HMI tags "Default tag table"
   "Clock_Byte" : Byte = PLC Clock_Byte AT %MB0, 100 ms
   "HMI_screenNumber" : Int = PLC HMI.screenNumber AT %DB1.DBW0, 100 ms
   "HMI_barcode" : Barcode Screen = PLC HMI.barcode AT %DB1.DBW0, 100 ms
   "HMI_partCall_current{0}" : Table Row = PLC HMI.partCall.current[0], 100 ms
   "HMI_partCall_current{1}" : Table Row = PLC HMI.partCall.current[1], 100 ms
   "HMI_partCall_current{2}" : Table Row = PLC HMI.partCall.current[2], 100 ms
   "HMI_partCall_current{3}" : Table Row = PLC HMI.partCall.current[3], 100 ms
   "HMI_partCall_current{4}" : Table Row = PLC HMI.partCall.current[4], 100 ms
   "HMI_partCall_current{5}" : Table Row = PLC HMI.partCall.current[5], 100 ms
   "HMI_partCall_current{6}" : Table Row = PLC HMI.partCall.current[6], 100 ms
   "HMI_partCall_current{7}" : Table Row = PLC HMI.partCall.current[7], 100 ms
   "HMI_partCall_current{8}" : Table Row = PLC HMI.partCall.current[8], 100 ms
   "HMI_partCall_current{9}" : Table Row = PLC HMI.partCall.current[9], 100 ms
   "HMI_partCall_current{10}" : Table Row = PLC HMI.partCall.current[10], 100 ms
   "HMI_settings_current_stations_selectBtns{0}" : PB Data: Text Label = PLC HMI.settings.current.stations.selectBtns[0], 100 ms
   "HMI_settings_current_stations_selectBtns{1}" : PB Data: Text Label = PLC HMI.settings.current.stations.selectBtns[1], 100 ms
   "HMI_settings_current_stations_selectBtns{2}" : PB Data: Text Label = PLC HMI.settings.current.stations.selectBtns[2], 100 ms
   "HMI_settings_current_stations_selectBtns{3}" : PB Data: Text Label = PLC HMI.settings.current.stations.selectBtns[3], 100 ms
   "HMI_settings_current_stations_selectBtns{4}" : PB Data: Text Label = PLC HMI.settings.current.stations.selectBtns[4], 100 ms
   "HMI_settings_current_stations_selectBtns{5}" : PB Data: Text Label = PLC HMI.settings.current.stations.selectBtns[5], 100 ms
   "HMI_settings_current_stations_selectBtns{6}" : PB Data: Text Label = PLC HMI.settings.current.stations.selectBtns[6], 100 ms
   "HMI_settings_current_stations_selectBtns{7}" : PB Data: Text Label = PLC HMI.settings.current.stations.selectBtns[7], 100 ms
   "HMI_settings_current_stations_selectBtns{8}" : PB Data: Text Label = PLC HMI.settings.current.stations.selectBtns[8], 100 ms
   "HMI_settings_current_stations_selectBtns{9}" : PB Data: Text Label = PLC HMI.settings.current.stations.selectBtns[9], 100 ms
   "HMI_settings_current_stations_selectBtns{10}" : PB Data: Text Label = PLC HMI.settings.current.stations.selectBtns[10], 100 ms
   "HMI_settings_current_stations_selectBtns{11}" : PB Data: Text Label = PLC HMI.settings.current.stations.selectBtns[11], 100 ms
   "HMI_settings_current_kp8_buttons{0}" : PB Data: Text Label = PLC HMI.settings.current.kp8.buttons[0], 100 ms
   "HMI_settings_current_kp8_buttons{7}" : PB Data: Text Label = PLC HMI.settings.current.kp8.buttons[7], 100 ms
   "HMI_settings_current_kp8_buttons{3}" : PB Data: Text Label = PLC HMI.settings.current.kp8.buttons[3], 100 ms
   "HMI_settings_current_kp8_buttons{6}" : PB Data: Text Label = PLC HMI.settings.current.kp8.buttons[6], 100 ms
   "HMI_settings_current_kp8_buttons{2}" : PB Data: Text Label = PLC HMI.settings.current.kp8.buttons[2], 100 ms
   "HMI_settings_current_kp8_buttons{5}" : PB Data: Text Label = PLC HMI.settings.current.kp8.buttons[5], 100 ms
   "HMI_settings_current_kp8_buttons{1}" : PB Data: Text Label = PLC HMI.settings.current.kp8.buttons[1], 100 ms
   "HMI_settings_current_kp8_buttons{4}" : PB Data: Text Label = PLC HMI.settings.current.kp8.buttons[4], 100 ms
   "HMI_settings_current_stations_selCount" : Int = PLC HMI.settings.current.stations.selCount, 100 ms
   "HMI_settings_current_viewingStation_btns{0}" : Station Assignment: Button Details = PLC HMI.settings.current.viewingStation.btns[0], 100 ms
   "HMI_settings_current_viewingStation_btns{1}" : Station Assignment: Button Details = PLC HMI.settings.current.viewingStation.btns[1], 100 ms
   "HMI_settings_current_viewingStation_btns{2}" : Station Assignment: Button Details = PLC HMI.settings.current.viewingStation.btns[2], 100 ms
   "HMI_settings_current_viewingStation_btns{3}" : Station Assignment: Button Details = PLC HMI.settings.current.viewingStation.btns[3], 100 ms
   "HMI_settings_current_viewingStation_btns{4}" : Station Assignment: Button Details = PLC HMI.settings.current.viewingStation.btns[4], 100 ms
   "HMI_settings_current_viewingStation_btns{5}" : Station Assignment: Button Details = PLC HMI.settings.current.viewingStation.btns[5], 100 ms
   "HMI_settings_current_viewingStation_previous" : PB Data: Graphic/Text List = PLC HMI.settings.current.viewingStation.previous, 100 ms
   "HMI_settings_current_viewingStation_next" : PB Data: Graphic/Text List = PLC HMI.settings.current.viewingStation.next, 100 ms
   "HMI_settings_current_stations_selectAll" : PB Data: Text Label = PLC HMI.settings.current.stations.selectAll, 100 ms
   "HMI_settings_current_partNumber_assign" : PB Data: Text Label = PLC HMI.settings.current.partNumber.assign, 100 ms
   "HMI_settings_current_partNumber_ioField" : IO Field Data: Part Number = PLC HMI.settings.current.partNumber.ioField, 100 ms
   "HMI_settings_current_alotted_assign" : PB Data: Text Label = PLC HMI.settings.current.alotted.assign, 100 ms
   "HMI_settings_current_alotted_ioField" : IO Field Data: Timers = PLC HMI.settings.current.alotted.ioField, 100 ms
   "HMI_settings_current_critical_assign" : PB Data: Text Label = PLC HMI.settings.current.critical.assign, 100 ms
   "HMI_settings_current_critical_ioField" : IO Field Data: Timers = PLC HMI.settings.current.critical.ioField, 100 ms
   "HMI_settings_current_kp8_selectButtons" : PB Data: Text Label = PLC HMI.settings.current.kp8.selectButtons, 100 ms
   "HMI_settings_current_viewingStation_dzData" : Drop Zone Data = PLC HMI.settings.current.viewingStation.dzData, 100 ms
   "HMI_settings_current_viewingStation_lineData" : Line Label Data = PLC HMI.settings.current.viewingStation.lineData, 100 ms
   "HMI_settings_current_stations_prevGroup" : PB Data: Graphic/Text List = PLC HMI.settings.current.stations.prevGroup, 100 ms
   "HMI_settings_current_stations_nextGroup" : PB Data: Graphic/Text List = PLC HMI.settings.current.stations.nextGroup, 100 ms
   "HMI_settings_current_viewingStation_name" : WString[20] = PLC HMI.settings.current.viewingStation.name, 100 ms

text list "Station Selection Single": 0 'Select a Station to View'; 1 'Assignments'

screen "1 PART CALL" 1366x768
   on GenerateScreen: SetTag("HMI_screenNumber", 1)
   Rectangle "Nav Panel 02" at 682,700 size 684x68
      Appearance <- "HMI_screenNumber"
   Rectangle "Nav Panel 01" at 0,700 size 685x68
      Appearance <- "HMI_screenNumber"
   Rectangle "Nav Panel 03 Top Border Hide" at 685,700 size 678x3
      Visibility <- "HMI_screenNumber"
   Rectangle "Nav Panel 01 Top Border Hide" at 3,700 size 679x3
      Visibility <- "HMI_screenNumber"
   Button "Settings Screen" at 683,700 size 683x68; TextOff 'SETTINGS'; Authorization "User administration"
      on Release: ActivateScreen("2 SETTINGS", 0)
   Button "Part Call Screen" at 0,700 size 683x68; TextOff 'PART CALL'
      on Release: ActivateScreen("1 PART CALL", 0)
   TextField "Header Line" at 32,32 size 216x53; Text 'LINE'
   TextField "Header Drop Zone" at 238,32 size 236x53; Text 'DROP ZONE'
   TextField "Header Part Number" at 474,32 size 648x53; Text 'PART NUMBER'
   TextField "Header Time" at 1112,32 size 222x53; Text 'TIME'
   ScreenModuleView "TableRow00" at 27,90 size 1312x52; ScreenModuleType ""
      Guid_{11997190-27688} <- "HMI_partCall_current{0}"
   ScreenModuleView "TableRow01" at 27,142 size 1312x52; ScreenModuleType ""
      Guid_{11997190-27688} <- "HMI_partCall_current{1}"
   ScreenModuleView "TableRow02" at 27,194 size 1312x52; ScreenModuleType ""
      Guid_{11997190-27688} <- "HMI_partCall_current{2}"
   ScreenModuleView "TableRow03" at 27,246 size 1312x52; ScreenModuleType ""
      Guid_{11997190-27688} <- "HMI_partCall_current{3}"
   ScreenModuleView "TableRow04" at 27,298 size 1312x52; ScreenModuleType ""
      Guid_{11997190-27688} <- "HMI_partCall_current{4}"
   ScreenModuleView "TableRow05" at 27,350 size 1312x52; ScreenModuleType ""
      Guid_{11997190-27688} <- "HMI_partCall_current{5}"
   ScreenModuleView "TableRow06" at 27,402 size 1312x52; ScreenModuleType ""
      Guid_{11997190-27688} <- "HMI_partCall_current{6}"
   ScreenModuleView "TableRow07" at 27,454 size 1312x52; ScreenModuleType ""
      Guid_{11997190-27688} <- "HMI_partCall_current{7}"
   ScreenModuleView "TableRow08" at 27,506 size 1312x52; ScreenModuleType ""
      Guid_{11997190-27688} <- "HMI_partCall_current{8}"
   ScreenModuleView "TableRow09" at 27,558 size 1312x52; ScreenModuleType ""
      Guid_{11997190-27688} <- "HMI_partCall_current{9}"
   ScreenModuleView "TableRow10" at 27,610 size 1312x52; ScreenModuleType ""
      Guid_{11997190-27688} <- "HMI_partCall_current{10}"

screen "2 SETTINGS" 1366x768
   on GenerateScreen: SetTag("HMI_screenNumber", 2)
   Rectangle "Part Call Nave Panel" at 0,700 size 685x68
      Appearance <- "HMI_screenNumber"
   Rectangle "Settings Nav Panel" at 682,700 size 684x68
      Appearance <- "HMI_screenNumber"
   Rectangle "Part Call Top Border Hide" at 3,700 size 679x3
      Visibility <- "HMI_screenNumber"
   Rectangle "Settings Top Border Hide" at 685,700 size 678x3
      Visibility <- "HMI_screenNumber"
   Button "Part Call Screen" at 0,700 size 683x68; TextOff 'PART CALL'
      on Release: ActivateScreen("1 PART CALL", 0)
   Button "Settings Screen" at 683,700 size 683x68; TextOff 'SETTINGS'
      on Release: ActivateScreen("2 SETTINGS", 0)
   Rectangle "Station Assignment Table BG Full" at 793,40 size 533x630
      Visibility <- "HMI_settings_current_stations_selCount"
   TextField "Current Station Single" at 803,50 size 513x45; Text 'Text'
      Visibility <- "HMI_settings_current_stations_selCount"
   TextField "Hide Line and Drop Zone Multi" at 803,101 size 513x40; Text 'select single station for Line and Drop Zone'
      Visibility <- "HMI_settings_current_stations_selCount"
   GraphicView "KP8 Image" at 496,247 size 275x412; Picture "kp8 image"
   Rectangle "Station Assignment Table BG Mini" at 793,40 size 533x65
      Visibility <- "HMI_settings_current_stations_selCount"
   ScreenModuleView "PB: Set PN" at 50,50 size 414x45; Guid_{11997190-63616} 'Assign Part Number'; ScreenModuleType ""
      Guid_{11997190-63605} <- "HMI_settings_current_partNumber_assign"
   ScreenModuleView "PN IO Field" at 50,100 size 414x50; ScreenModuleType ""
      Guid_{11997190-63113} <- "HMI_settings_current_partNumber_ioField"
   ScreenModuleView "PB: Set Allotted" at 494,50 size 137x45; Guid_{11997190-63616} 'Allotted'; ScreenModuleType ""
      Guid_{11997190-63605} <- "HMI_settings_current_alotted_assign"
   ScreenModuleView "PB: Set Critical" at 636,50 size 137x45; Guid_{11997190-63616} 'Crititcal'; ScreenModuleType ""
      Guid_{11997190-63605} <- "HMI_settings_current_critical_assign"
   ScreenModuleView "Alotted Time IO Field" at 494,100 size 137x50; ScreenModuleType ""
      Guid_{11997190-63269} <- "HMI_settings_current_alotted_ioField"
   ScreenModuleView "Critical Time IO Field" at 636,100 size 137x50; ScreenModuleType ""
      Guid_{11997190-63269} <- "HMI_settings_current_critical_ioField"
   ScreenModuleView "PB: Select KP8 Buttons" at 493,190 size 284x45; Guid_{11997190-63616} 'Select Buttons'; ScreenModuleType ""
      Guid_{11997190-63605} <- "HMI_settings_current_kp8_selectButtons"
   ScreenModuleView "KP8 00: RESET" at 641,534 size 68x66; ScreenModuleType ""
      Guid_{11997190-57808} <- "HMI_settings_current_kp8_buttons{0}"
   ScreenModuleView "KP8 01" at 641,455 size 68x66; ScreenModuleType ""
      Guid_{11997190-57808} <- "HMI_settings_current_kp8_buttons{1}"
   ScreenModuleView "KP8 02" at 641,379 size 68x66; ScreenModuleType ""
      Guid_{11997190-57808} <- "HMI_settings_current_kp8_buttons{2}"
   ScreenModuleView "KP8 03" at 641,303 size 68x66; ScreenModuleType ""
      Guid_{11997190-57808} <- "HMI_settings_current_kp8_buttons{3}"
   ScreenModuleView "KP8 04: STOP RUNTIME" at 557,534 size 68x66; ScreenModuleType ""
      on Guid_{11997190-59171}: StopRuntime(0)
      Guid_{11997190-57808} <- "HMI_settings_current_kp8_buttons{4}"
   ScreenModuleView "KP8 05" at 557,455 size 68x66; ScreenModuleType ""
      Guid_{11997190-57808} <- "HMI_settings_current_kp8_buttons{5}"
   ScreenModuleView "KP8 06" at 557,379 size 68x66; ScreenModuleType ""
      Guid_{11997190-57808} <- "HMI_settings_current_kp8_buttons{6}"
   ScreenModuleView "KP8 07" at 557,303 size 68x66; ScreenModuleType ""
      Guid_{11997190-57808} <- "HMI_settings_current_kp8_buttons{7}"
   ScreenModuleView "PB: Previous Group" at 50,190 size 65x45; Guid_{11997190-63799} "Graphic_4"; ScreenModuleType ""
      Guid_{11997190-63779} <- "HMI_settings_current_stations_prevGroup"
   ScreenModuleView "PB: Select All Stations" at 120,190 size 274x45; Guid_{11997190-63616} 'Select Stations'; ScreenModuleType ""
      Guid_{11997190-63605} <- "HMI_settings_current_stations_selectAll"
   ScreenModuleView "PB: Next Group" at 399,190 size 65x45; Guid_{11997190-63799} "Graphic_3"; ScreenModuleType ""
      Guid_{11997190-63779} <- "HMI_settings_current_stations_nextGroup"
   ScreenModuleView "Station 00 Select" at 50,240 size 205x65; ScreenModuleType ""
      Guid_{11997190-57808} <- "HMI_settings_current_stations_selectBtns{0}"
   ScreenModuleView "Station 01 Select" at 260,240 size 205x65; ScreenModuleType ""
      Guid_{11997190-57808} <- "HMI_settings_current_stations_selectBtns{1}"
   ScreenModuleView "Station 02 Select" at 50,311 size 205x65; ScreenModuleType ""
      Guid_{11997190-57808} <- "HMI_settings_current_stations_selectBtns{2}"
   ScreenModuleView "Station 03 Select" at 260,311 size 205x65; ScreenModuleType ""
      Guid_{11997190-57808} <- "HMI_settings_current_stations_selectBtns{3}"
   ScreenModuleView "Station 04 Select" at 50,382 size 205x65; ScreenModuleType ""
      Guid_{11997190-57808} <- "HMI_settings_current_stations_selectBtns{4}"
   ScreenModuleView "Station 05 Select" at 260,382 size 205x65; ScreenModuleType ""
      Guid_{11997190-57808} <- "HMI_settings_current_stations_selectBtns{5}"
   ScreenModuleView "Station 06 Select" at 50,453 size 205x65; ScreenModuleType ""
      Guid_{11997190-57808} <- "HMI_settings_current_stations_selectBtns{6}"
   ScreenModuleView "Station 07 Select" at 260,453 size 205x65; ScreenModuleType ""
      Guid_{11997190-57808} <- "HMI_settings_current_stations_selectBtns{7}"
   ScreenModuleView "Station 08 Select" at 50,524 size 205x65; ScreenModuleType ""
      Guid_{11997190-57808} <- "HMI_settings_current_stations_selectBtns{8}"
   ScreenModuleView "Station 09 Select" at 260,524 size 205x65; ScreenModuleType ""
      Guid_{11997190-57808} <- "HMI_settings_current_stations_selectBtns{9}"
   ScreenModuleView "Station 10 Select" at 50,595 size 205x65; ScreenModuleType ""
      Guid_{11997190-57808} <- "HMI_settings_current_stations_selectBtns{10}"
   ScreenModuleView "Station 11 Select" at 260,595 size 205x65; ScreenModuleType ""
      Guid_{11997190-57808} <- "HMI_settings_current_stations_selectBtns{11}"
   ScreenModuleView "Line Label" at 803,101 size 267x40; ScreenModuleType ""
      Guid_{11997190-64598} <- "HMI_settings_current_viewingStation_lineData"
   ScreenModuleView "Drop Zone Label" at 1076,101 size 240x40; ScreenModuleType ""
      Guid_{11997190-64802} <- "HMI_settings_current_viewingStation_dzData"
   ScreenModuleView "PB: Previous Station" at 803,50 size 65x45; Guid_{11997190-63799} "Graphic_1"; ScreenModuleType ""
      Guid_{11997190-63779} <- "HMI_settings_current_viewingStation_previous"
   TextField "Current Station Multi" at 873,50 size 373x45; Text 'Assignments'
      Visibility <- "HMI_settings_current_stations_selCount"
   ScreenModuleView "PB: Next Station" at 1251,50 size 65x45; Guid_{11997190-63799} "Graphic_2"; ScreenModuleType ""
      Guid_{11997190-63779} <- "HMI_settings_current_viewingStation_previous"
   TextField "Button Column Header" at 803,146 size 75x40; Text 'Btn'
      Visibility <- "HMI_settings_current_stations_selCount"
   TextField "Timer Column Header" at 872,146 size 128x40; Text 'Times'
      Visibility <- "HMI_settings_current_stations_selCount"
   TextField "Part Number Column Header" at 993,146 size 323x40; Text 'Part Number'
      Visibility <- "HMI_settings_current_stations_selCount"
   ScreenModuleView "Button 00 Details" at 803,191 size 513x74; ScreenModuleType ""
      Guid_{11997190-60358} <- "HMI_settings_current_viewingStation_btns{0}"
   ScreenModuleView "Button 01 Details" at 803,270 size 513x74; ScreenModuleType ""
      Guid_{11997190-60358} <- "HMI_settings_current_viewingStation_btns{1}"
   ScreenModuleView "Button 02 Details" at 803,349 size 513x74; ScreenModuleType ""
      Guid_{11997190-60358} <- "HMI_settings_current_viewingStation_btns{2}"
   ScreenModuleView "Button 03 Details" at 803,428 size 513x74; ScreenModuleType ""
      Guid_{11997190-60358} <- "HMI_settings_current_viewingStation_btns{3}"
   ScreenModuleView "Button 04 Details" at 803,507 size 513x74; ScreenModuleType ""
      Guid_{11997190-60358} <- "HMI_settings_current_viewingStation_btns{4}"
   ScreenModuleView "Button 05 Details" at 803,586 size 513x74; ScreenModuleType ""
      Guid_{11997190-60358} <- "HMI_settings_current_viewingStation_btns{5}"

screen "3 BARCODE" 1366x768
   on GenerateScreen: SetTag("HMI_screenNumber", 3)
   Rectangle "Nav Panel 02" at 682,700 size 684x68
      Appearance <- "HMI_screenNumber"
   Rectangle "Nav Panel 01" at 0,700 size 685x68
      Appearance <- "HMI_screenNumber"
   Rectangle "Nav Panel 03 Top Border Hide" at 685,700 size 678x3
      Visibility <- "HMI_screenNumber"
   Rectangle "Nav Panel 01 Top Border Hide" at 3,700 size 679x3
      Visibility <- "HMI_screenNumber"
   Button "Settings Screen" at 683,700 size 683x68; TextOff 'SETTINGS'; Authorization "User administration"
      on Release: ActivateScreen("2 SETTINGS", 0)
   Button "Part Call Screen" at 0,700 size 683x68; TextOff 'PART CALL'
      on Release: ActivateScreen("1 PART CALL", 0)
   Button "btCancel" at 685,431 size 649x68; TextOff 'CANCEL'
      on Release: ActivateScreen("1 PART CALL", 0)
   Button "btPartOrdered" at 32,431 size 648x68; TextOff 'ORDERED'
      on Release: SetBit("ordered"); ActivateScreen("1 PART CALL", 0)
   TextField "tfBarcodeDisplay" at 32,220 size 1302x206; Text 'Text'
   TextField "tfPartNumberDisplay" at 32,160 size 1302x53; Text 'BARCODE FOR PART NUMBER'
*)

(* ===== HMI "HMI_RT_2" =====
connection "HMI_Connection_3": ETHERNET, S7_1500_OMS

HMI tags "Default tag table"
   "Clock_0.5Hz" : Bool = PLC "Clock_0.5Hz" AT %M0.7, 100 ms
   "LED Sign_request_row{0}" : Table Row = PLC "LED Sign".request.row[0], 1 s
   "LED Sign_request_row{1}" : Table Row = PLC "LED Sign".request.row[1], 1 s
   "LED Sign_request_row{2}" : Table Row = PLC "LED Sign".request.row[2], 1 s
   "LED Sign_request_row{3}" : Table Row = PLC "LED Sign".request.row[3], 1 s
   "LED Sign_request_row{4}" : Table Row = PLC "LED Sign".request.row[4], 1 s
   "LED Sign_request_row{5}" : Table Row = PLC "LED Sign".request.row[5], 1 s
   "LED Sign_request_row{6}" : Table Row = PLC "LED Sign".request.row[6], 1 s
   "LED Sign_request_row{7}" : Table Row = PLC "LED Sign".request.row[7], 1 s
   "LED Sign_request_row{8}" : Table Row = PLC "LED Sign".request.row[8], 1 s
   "LED Sign_request_row{9}" : Table Row = PLC "LED Sign".request.row[9], 1 s
   "LED Sign_request_row{10}" : Table Row = PLC "LED Sign".request.row[10], 1 s
   "LED Sign_request_row{11}" : Table Row = PLC "LED Sign".request.row[11], 1 s

screen "1 PART CALL" 1024x768
   Rectangle "Connection Status" at 1,196 size 894x1
      Appearance <- "Clock_0.5Hz"
   ScreenModuleView "R0C0" at 6,9 size 440x28; ScreenModuleType ""
      Guid_{11997190-27688} <- "LED Sign_request_row{0}"
   ScreenModuleView "R1C0" at 6,39 size 440x28; ScreenModuleType ""
      Guid_{11997190-27688} <- "LED Sign_request_row{1}"
   ScreenModuleView "R2C0" at 6,69 size 440x28; ScreenModuleType ""
      Guid_{11997190-27688} <- "LED Sign_request_row{2}"
   ScreenModuleView "R3C0" at 6,99 size 440x28; ScreenModuleType ""
      Guid_{11997190-27688} <- "LED Sign_request_row{3}"
   ScreenModuleView "R4C0" at 6,128 size 440x28; ScreenModuleType ""
      Guid_{11997190-27688} <- "LED Sign_request_row{4}"
   ScreenModuleView "R5C0" at 6,158 size 440x28; ScreenModuleType ""
      Guid_{11997190-27688} <- "LED Sign_request_row{5}"
   ScreenModuleView "R0C1" at 455,9 size 438x28; ScreenModuleType ""
      Guid_{11997190-27688} <- "LED Sign_request_row{6}"
   ScreenModuleView "R1C1" at 455,39 size 438x28; ScreenModuleType ""
      Guid_{11997190-27688} <- "LED Sign_request_row{7}"
   ScreenModuleView "R2C1" at 454,69 size 440x28; ScreenModuleType ""
      Guid_{11997190-27688} <- "LED Sign_request_row{8}"
   ScreenModuleView "R3C1" at 454,99 size 440x28; ScreenModuleType ""
      Guid_{11997190-27688} <- "LED Sign_request_row{9}"
   ScreenModuleView "R4C1" at 454,128 size 440x28; ScreenModuleType ""
      Guid_{11997190-27688} <- "LED Sign_request_row{10}"
   ScreenModuleView "R5C1" at 454,158 size 440x28; ScreenModuleType ""
      Guid_{11997190-27688} <- "LED Sign_request_row{11}"
*)

(* ===== HMI "HMI_RT_1" =====
system functions are stored by id; their names below are inferred from use

ScreenModuleEditorView "Table Row" 1312x52
   TextField "tfLine" at 5,1 size 216x48; Text 'Text'
      Visibility <- "interface.tfLine.visibility"
      Appearance <- "interface.tfLine.animator"
   TextField "tfTime" at 1085,1 size 222x48; Text 'Text'
      Appearance <- "interface.tfTime.animator"
      Visibility <- "interface.tfTime.visibility"
   TextField "tfDropZone" at 211,1 size 236x48; Text 'Text'
      Appearance <- "interface.tfDropZone.animator"
      Visibility <- "interface.tfDropZone.visibility"
   TextField "tfPartNumber" at 445,1 size 650x48; Text 'Text'
      Appearance <- "interface.tfPartNumber.animator"
      Visibility <- "interface.tfPartNumber.visibility"
   Button "pbSelect" at 0,0 size 1312x52; TextOff 'Text'
      Visibility <- "interface.pbSelection.visibility"
      on Press: SetBit("interface.pbSelection.request")
      on Release: ResetBit("interface.pbSelection.request")
   Rectangle "rtBackground" at 0,0 size 1312x52
      Visibility <- "interface.rtBackground.visibility"
*)

(* ===== HMI "HMI_RT_1" =====
system functions are stored by id; their names below are inferred from use

ScreenModuleEditorView "Table Row" 1312x52
   TextField "tfLine" at 5,1 size 216x48; Text 'Text'
      Visibility <- "interface.tfLine.visibility"
      Appearance <- "interface.tfLine.animator"
   TextField "tfTime" at 1085,1 size 222x48; Text 'Text'
      Visibility <- "interface.tfTime.visibility"
      Appearance <- "interface.tfTime.animator"
   TextField "tfDropZone" at 211,1 size 236x48; Text 'Text'
      Visibility <- "interface.tfDropZone.visibility"
      Appearance <- "interface.tfDropZone.animator"
   TextField "tfPartNumber" at 445,1 size 650x48; Text 'Text'
      Visibility <- "interface.tfPartNumber.visibility"
      Appearance <- "interface.tfPartNumber.animator"
   Button "pbSelect" at 0,0 size 1312x52; TextOff 'Text'
      on Release: ResetBit("interface.pbSelection.request")
      on Press: SetBit("interface.pbSelection.request")
      Visibility <- "interface.pbSelection.visibility"
   Rectangle "rtBackground" at 0,0 size 1312x52
      Visibility <- "interface.rtBackground.visibility"
*)

(* ===== HMI "HMI_RT_1" =====
system functions are stored by id; their names below are inferred from use

ScreenModuleEditorView "Table Row" 1312x52
   TextField "tfLine" at 5,1 size 216x48; Text 'Text'
      Visibility <- "interface.tfLine.visibility"
      Appearance <- "interface.tfLine.animator"
   TextField "tfTime" at 1085,1 size 222x48; Text 'Text'
      Visibility <- "interface.tfTime.visibility"
      Appearance <- "interface.tfTime.animator"
   TextField "tfDropZone" at 211,1 size 236x48; Text 'Text'
      Visibility <- "interface.tfDropZone.visibility"
      Appearance <- "interface.tfDropZone.animator"
   TextField "tfPartNumber" at 445,1 size 650x48; Text 'Text'
      Visibility <- "interface.tfPartNumber.visibility"
      Appearance <- "interface.tfPartNumber.animator"
   Button "pbSelect" at 0,0 size 1312x52; TextOff 'Text'
      on Release: ResetBit("interface.pbSelection.request")
      on Press: SetBit("interface.pbSelection.request")
      Visibility <- "interface.pbSelection.visibility"
   Rectangle "rtBackground" at 0,0 size 1312x52
      Visibility <- "interface.rtBackground.visibility"
*)

(* ===== HMI "HMI_RT_1" =====
system functions are stored by id; their names below are inferred from use

ScreenModuleEditorView "Table Row" 1312x52
   TextField "tfLine" at 5,1 size 216x48; Text 'Text'
      Visibility <- "interface.tfLine.visibility"
      Appearance <- "interface.tfLine.animator"
   TextField "tfTime" at 1085,1 size 222x48; Text 'Text'
      Visibility <- "interface.tfTime.visibility"
      Appearance <- "interface.tfTime.animator"
   TextField "tfDropZone" at 211,1 size 236x48; Text 'Text'
      Visibility <- "interface.tfDropZone.visibility"
      Appearance <- "interface.tfDropZone.animator"
   TextField "tfPartNumber" at 445,1 size 650x48; Text 'Text'
      Visibility <- "interface.tfPartNumber.visibility"
      Appearance <- "interface.tfPartNumber.animator"
   Button "pbSelect" at 0,0 size 1312x52; TextOff 'Text'
      on Release: ResetBit("interface.pbSelection.request")
      on Press: SetBit("interface.pbSelection.request")
      Visibility <- "interface.pbSelection.visibility"
   Rectangle "rtBackground" at 0,0 size 1312x52
      Visibility <- "interface.rtBackground.visibility"
*)

(* ===== HMI "HMI_RT_1" =====
system functions are stored by id; their names below are inferred from use

ScreenModuleEditorView "Table Row" 1312x52
   TextField "tfLine" at 5,1 size 216x48; Text 'Text'
      Visibility <- "interface.tfLine.visibility"
      Appearance <- "interface.tfLine.animator"
   TextField "tfTime" at 1085,1 size 222x48; Text 'Text'
      Visibility <- "interface.tfTime.visibility"
      Appearance <- "interface.tfTime.animator"
   TextField "tfDropZone" at 211,1 size 236x48; Text 'Text'
      Visibility <- "interface.tfDropZone.visibility"
      Appearance <- "interface.tfDropZone.animator"
   TextField "tfPartNumber" at 445,1 size 650x48; Text 'Text'
      Visibility <- "interface.tfPartNumber.visibility"
      Appearance <- "interface.tfPartNumber.animator"
   Button "pbSelect" at 0,0 size 1312x52; TextOff 'Text'
      on Release: ResetBit("interface.pbSelection.request")
      on Press: SetBit("interface.pbSelection.request")
      Visibility <- "interface.pbSelection.visibility"
   Rectangle "rtBackground" at 0,0 size 1312x52
      Visibility <- "interface.rtBackground.visibility"
*)

(* ===== HMI "HMI_RT_1" =====
system functions are stored by id; their names below are inferred from use

ScreenModuleEditorView "LED Row" 1312x52
   TextField "tfLine" at 5,1 size 216x48; Text 'Text'
      Visibility <- "interface.tfLine.visibility"
      Appearance <- "interface.tfLine.animator"
   TextField "tfTime" at 1085,1 size 222x48; Text 'Text'
      Visibility <- "interface.tfTime.visibility"
      Appearance <- "interface.tfTime.animator"
   TextField "tfDropZone" at 211,1 size 236x48; Text 'Text'
      Visibility <- "interface.tfDropZone.visibility"
      Appearance <- "interface.tfDropZone.animator"
   TextField "tfPartNumber" at 445,1 size 650x48; Text 'Text'
      Visibility <- "interface.tfPartNumber.visibility"
      Appearance <- "interface.tfPartNumber.animator"
   Button "pbSelect" at 0,0 size 1312x52; TextOff 'Text'
      on Release: ResetBit("interface.pbSelection.request")
      on Press: SetBit("interface.pbSelection.request")
      Visibility <- "interface.pbSelection.visibility"
   Rectangle "rtBackground" at 0,0 size 1312x52
      Visibility <- "interface.rtBackground.visibility"
*)

(* ===== HMI "HMI_RT_1" =====
system functions are stored by id; their names below are inferred from use

ScreenModuleEditorView "LED Row" 440x28
   TextField "tfLine" at 0,0 size 110x28; Text 'Text'
      Visibility <- "interface.tfLine.visibility"
      Appearance <- "interface.tfLine.animator"
   TextField "tfTime" at 349,0 size 91x28; Text 'Text'
      Visibility <- "interface.tfTime.visibility"
      Appearance <- "interface.tfTime.animator"
   TextField "tfDropZone" at 105,0 size 42x28; Text 'Text'
      Visibility <- "interface.tfDropZone.visibility"
      Appearance <- "interface.tfDropZone.animator"
   TextField "tfDLPartNumber" at 146,0 size 209x28; Text 'Text'
      Appearance <- "interface.tfPartNumber.animator"
      Visibility <- "interface.tfPartNumber.count"
   Button "pbSelect" at 0,0 size 440x28; TextOff 'Text'
      on Release: ResetBit("interface.pbSelection.request")
      on Press: SetBit("interface.pbSelection.request")
      Visibility <- "interface.pbSelection.visibility"
   Rectangle "rtBackground" at 0,0 size 440x28
      Visibility <- "interface.rtBackground.visibility"
   TextField "tfSLPartNumber" at 146,0 size 209x28; Text 'Text'
      Appearance <- "interface.tfPartNumber.animator"
      Visibility <- "interface.tfPartNumber.count"
*)

(* ===== HMI "HMI_RT_1" =====
system functions are stored by id; their names below are inferred from use

ScreenModuleEditorView "Table Row" 1312x52
   TextField "tfLine" at 5,1 size 216x48; Text 'Text'
      Visibility <- "interface.tfLine.visibility"
      Appearance <- "interface.tfLine.animator"
   TextField "tfTime" at 1085,1 size 222x48; Text 'Text'
      Visibility <- "interface.tfTime.visibility"
      Appearance <- "interface.tfTime.animator"
   TextField "tfDropZone" at 211,1 size 236x48; Text 'Text'
      Visibility <- "interface.tfDropZone.visibility"
      Appearance <- "interface.tfDropZone.animator"
   TextField "tfSLPartNumber" at 445,1 size 650x48; Text 'Text'
      Appearance <- "interface.tfPartNumber.animator"
      Visibility <- "interface.tfPartNumber.count"
   Button "pbSelect" at 0,0 size 1312x52; TextOff 'Text'
      on Release: ResetBit("interface.pbSelection.request")
      on Press: SetBit("interface.pbSelection.request")
      Visibility <- "interface.pbSelection.visibility"
   Rectangle "rtBackground" at 0,0 size 1312x52
      Visibility <- "interface.rtBackground.visibility"
   TextField "tfDLPartNumber" at 445,1 size 650x48; Text 'Text'
      Appearance <- "interface.tfPartNumber.animator"
      Visibility <- "interface.tfPartNumber.count"
*)

(* ===== HMI "HMI_RT_1" =====

ScreenModuleEditorView "LED Row" 440x28
   TextField "tfLine" at 0,0 size 110x28; Text 'Text'
      Visibility <- "interface.tfLine.visibility"
      Appearance <- "interface.tfLine.animator"
   TextField "tfTime" at 349,0 size 91x28; Text 'Text'
      Visibility <- "interface.tfTime.visibility"
      Appearance <- "interface.tfTime.animator"
   TextField "tfDropZone" at 105,0 size 42x28; Text 'Text'
      Visibility <- "interface.tfDropZone.visibility"
      Appearance <- "interface.tfDropZone.animator"
   TextField "tfSLPartNumber" at 146,0 size 209x28; Text 'Text'
      Visibility <- "interface.tfPartNumber.count"
      Appearance <- "interface.tfPartNumber.animator"
   TextField "tfDLPartNumber" at 146,0 size 209x28; Text 'Text'
      Visibility <- "interface.tfPartNumber.count"
      Appearance <- "interface.tfPartNumber.animator"
*)

(* ===== HMI "HMI_RT_1" =====
system functions are stored by id; their names below are inferred from use

ScreenModuleEditorView "Table Row" 1312x52
   TextField "tfLine" at 5,1 size 216x48; Text 'Text'
      Visibility <- "interface.tfLine.visibility"
      Appearance <- "interface.tfLine.animator"
   TextField "tfTime" at 1085,1 size 222x48; Text 'Text'
      Visibility <- "interface.tfTime.visibility"
      Appearance <- "interface.tfTime.animator"
   TextField "tfDropZone" at 211,1 size 236x48; Text 'Text'
      Visibility <- "interface.tfDropZone.visibility"
      Appearance <- "interface.tfDropZone.animator"
   TextField "tfSLPartNumber" at 445,1 size 650x48; Text 'Text'
      Visibility <- "interface.tfPartNumber.count"
      Appearance <- "interface.tfPartNumber.animator"
   Button "pbSelect" at 0,0 size 1312x52; TextOff 'Text'
      on Release: ResetBit("interface.pbSelection.request")
      on Press: SetBit("interface.pbSelection.request")
      Visibility <- "interface.pbSelection.visibility"
   Rectangle "rtBackground" at 0,0 size 1312x52
      Visibility <- "interface.rtBackground.visibility"
   TextField "tfDLPartNumber" at 445,1 size 650x48; Text 'Text'
      Visibility <- "interface.tfPartNumber.count"
      Appearance <- "interface.tfPartNumber.animator"
*)

(* ===== HMI "HMI_RT_1" =====
system functions are stored by id; their names below are inferred from use

ScreenModuleEditorView "PB: Station Select (Text Label)" 205x65
   Button "Station Select" at 0,0 size 205x65; TextOff 'Text'
      on Press: function_b14e0dd5("Interface.actuate", 0)
      Appearance <- "Interface.animate"
*)

(* ===== HMI "HMI_RT_1" =====
system functions are stored by id; their names below are inferred from use

ScreenModuleEditorView "PB: KP8 Button Select (Text Label)" 205x65
   Button "Station Select" at 0,0 size 205x65; TextOff 'Text'
      on Press: function_b14e0dd5("Interface.actuate", 0)
      Appearance <- "Interface.animate"
*)

(* ===== HMI "HMI_RT_1" =====
system functions are stored by id; their names below are inferred from use

ScreenModuleEditorView "PB: KP8 Button Select (Text Label)" 68x66
   Button "Station Select" at 0,0 size 68x66; TextOff 'Text'
      on Press: function_b14e0dd5("Interface.actuate", 0)
      Appearance <- "Interface.animate"
*)

(* ===== HMI "HMI_RT_1" =====
system functions are stored by id; their names below are inferred from use

ScreenModuleEditorView "PB: KP8 Stop Runtime (Text Label)" 68x66
   Button "Station Select" at 0,0 size 68x66; TextOff 'Text'
      on Press: function_b14e0dd5("Interface.actuate", 0)
      Appearance <- "Interface.animate"
*)

(* ===== HMI "HMI_RT_1" =====

ScreenModuleEditorView "PB: KP8 Stop Runtime (Text Label)" 68x66
   Button "Station Select" at 0,0 size 68x66; TextOff 'NOT USED'
      Appearance <- "Interface.animate"
*)

(* ===== HMI "HMI_RT_1" =====

ScreenModuleEditorView "PB: KP8 Stop Runtime (Text Label)" 68x66
   Button "Station Select" at 0,0 size 68x66; TextOff 'NOT USED'
      Appearance <- "Interface.animate"
*)

(* ===== HMI "HMI_RT_1" =====
system functions are stored by id; their names below are inferred from use

ScreenModuleEditorView "Station Assignment: Button Details" 513x74
   TextField "Button Label" at 0,0 size 75x74; Text 'Text'
      Appearance <- "Interface.label.animate"
      Visibility <- "Interface.label.animate"
   TextField "Critical Time" at 70,37 size 122x37; Text 'Text'
      Appearance <- "Interface.critical.animate"
      Visibility <- "Interface.critical.animate"
   TextField "Alloted Time" at 70,0 size 122x38; Text 'Text'
      Appearance <- "Interface.alloted.animate"
      Visibility <- "Interface.alloted.animate"
   TextField "Part Number" at 185,0 size 328x74; Text 'Text'
      Appearance <- "Interface.partNumber.animate"
      Visibility <- "Interface.partNumber.animate"
   Button "Select PB" at 0,0 size 513x74; TextOff 'Text'
      on Press: function_b14e0dd5("Interface.select.actuate", 0)
      Visibility <- "Interface.select.animate"
      ObjectEnable <- "Interface.select.animate"
*)

(* ===== HMI "HMI_RT_1" =====
system functions are stored by id; their names below are inferred from use

ScreenModuleEditorView "IO Field: Part Number" 414x50
   IOField "PN Entry Field" at 0,0 size 414x50; FormatPattern ????????????????????????????????????????
      on OnFinishInput: SetBit("Interface.inputFinished")
      ObjectEnable <- "Interface.animate"
      Appearance <- "Interface.animate"
      ProcessValue <- "Interface.value"
*)

(* ===== HMI "HMI_RT_1" =====
system functions are stored by id; their names below are inferred from use

ScreenModuleEditorView "IO Field: Timer" 137x50
   IOField "Allotted Time Entry Field" at 0,0 size 137x50; FormatPattern ???????
      Appearance <- "Interface.animate"
      ObjectEnable <- "Interface.animate"
      on OnFinishInput: SetBit("Interface.inputFinished")
      ProcessValue <- "Interface.value"
*)

(* ===== HMI "HMI_RT_1" =====
system functions are stored by id; their names below are inferred from use

ScreenModuleEditorView "PB: Text Label" 274x45
   Button "Select All Stations" at 0,0 size 274x45; TextOff 'Text'
      on Press: function_b14e0dd5("Interface.actuate", 0)
      Appearance <- "Interface.animate"
*)

(* ===== HMI "HMI_RT_1" =====
system functions are stored by id; their names below are inferred from use

ScreenModuleEditorView "PB: Graphic/Text List" 65x45
   Button "Previous Station Group" at 0,0 size 65x45; TextOff 'Text'
      Visibility <- "Interface.animate"
      ObjectEnable <- "Interface.animate"
      Appearance <- "Interface.animate"
      on Press: SetBit("Interface.actuate")
*)

(* ===== HMI "HMI_RT_1" =====
system functions are stored by id; their names below are inferred from use

ScreenModuleEditorView "Line Label" 267x40
   IOField "Line" at 86,0 size 181x40; FormatPattern ?????????
      Appearance <- "interface.animate.ioField"
      ObjectEnable <- "interface.animate.ioField"
      Visibility <- "interface.animate.ioField"
      on OnFinishInput: SetBit("interface.inputFinished")
      ProcessValue <- "interface.value"
   TextField "Line Label" at 0,0 size 267x40; Text 'Line:'
      Appearance <- "interface.animate.bg"
      Visibility <- "interface.animate.bg"
*)

(* ===== HMI "HMI_RT_1" =====
system functions are stored by id; their names below are inferred from use

ScreenModuleEditorView "Drop Zone Label" 240x40
   IOField "Drop Zone Entry" at 171,0 size 69x40; FormatPattern ??
      Appearance <- "Interface.animate.ioField"
      ObjectEnable <- "Interface.animate.ioField"
      Visibility <- "Interface.animate.ioField"
      on OnFinishInput: SetBit("Interface.inputFinished")
      ProcessValue <- "Interface.value"
   TextField "Drop Zone Label" at 0,0 size 240x40; Text 'Drop Zone:'
      Appearance <- "Interface.animate.bg"
      Visibility <- "Interface.animate.bg"
*)

(* ===== HMI "HMI_RT_1" =====

ScreenModuleEditorView "PB: KP8 Reset Button (Text Label" 68x66
   Button "Station Select" at 0,0 size 68x66; TextOff 'NOT USED'
      Appearance <- "Interface.animate"
*)

(* ===== HMI "HMI_RT_1" =====

ScreenModuleEditorView "PB: KP8 Reset Button (Text Label" 68x66
   Button "Station Select" at 0,0 size 68x66; TextOff 'RESET SELECTED'
      Appearance <- "Interface.animate"
*)

(* ===== HMI "HMI_RT_1" =====

ScreenModuleEditorView "PB: KP8 Stop Runtime (Text Label)" 68x66
   Button "Station Select" at 0,0 size 68x66; TextOff 'STOP RUNTIME'
      Appearance <- "Interface.animate"
*)

(* ===== HMI "HMI_RT_1" =====
system functions are stored by id; their names below are inferred from use

ScreenModuleEditorView "PB: Graphic/Text List" 65x45
   Button "Previous Station Group" at 0,0 size 65x45; TextOff 'Text'
      on Press: SetBit("Interface.actuate")
      Visibility <- "Interface.animate"
      ObjectEnable <- "Interface.animate"
      Appearance <- "Interface.animate"
*)

(* ===== HMI "HMI_RT_1" =====
system functions are stored by id; their names below are inferred from use

ScreenModuleEditorView "PB: Text Label" 274x45
   Button "Select All Stations" at 0,0 size 274x45; TextOff 'Text'
      on Press: function_b14e0dd5("Interface.actuate", 0)
      Appearance <- "Interface.animate"
*)

(* ===== HMI "HMI_RT_1" =====
system functions are stored by id; their names below are inferred from use

ScreenModuleEditorView "PB: Text Label" 274x45
   Button "Select All Stations" at 0,0 size 274x45; TextOff 'Text'
      on Press: function_b14e0dd5("Interface.actuate", 0)
      Appearance <- "Interface.animate"
*)

(* ===== HMI "HMI_RT_1" =====
system functions are stored by id; their names below are inferred from use

ScreenModuleEditorView "PB: Graphic/Text List" 65x45
   Button "Previous Station Group" at 0,0 size 65x45; TextOff 'Text'
      on Press: SetBit("Interface.actuate")
      Visibility <- "Interface.animate"
      ObjectEnable <- "Interface.animate"
      Appearance <- "Interface.animate"
*)

(* ===== HMI "HMI_RT_1" =====
system functions are stored by id; their names below are inferred from use

ScreenModuleEditorView "PB: Station Select (Text Label)" 205x65
   Button "Station Select" at 0,0 size 205x65; TextOff 'Text'
      on Press: function_b14e0dd5("Interface.actuate", 0)
      Appearance <- "Interface.animate"
*)

(* ===== HMI "HMI_RT_1" =====
system functions are stored by id; their names below are inferred from use

ScreenModuleEditorView "PB: Graphic/Text List" 65x45
   Button "Previous Station Group" at 0,0 size 65x45; TextOff 'Text'
      on Press: function_b14e0dd5("Interface.actuate", 0)
      Visibility <- "Interface.animate"
      ObjectEnable <- "Interface.animate"
      Appearance <- "Interface.animate"
*)

(* ===== HMI "HMI_RT_1" =====
system functions are stored by id; their names below are inferred from use

ScreenModuleEditorView "Drop Zone Label" 240x40
   IOField "Drop Zone Entry" at 171,0 size 69x40; FormatPattern ??
      on OnFinishInput: SetBit("Interface.inputFinished")
      Appearance <- "Interface.animate.ioField"
      ObjectEnable <- "Interface.animate.ioField"
      Visibility <- "Interface.animate.ioField"
      ProcessValue <- "Interface.value"
   TextField "Drop Zone Label" at 0,0 size 240x40; Text 'Drop Zone:'
      Visibility <- "Interface.animate.bg"
      Appearance <- "Interface.animate.bg"
*)

(* ===== HMI "HMI_RT_1" =====
system functions are stored by id; their names below are inferred from use

ScreenModuleEditorView "IO Field: Part Number" 414x50
   IOField "PN Entry Field" at 0,0 size 414x50; FormatPattern ????????????????????????????????????????
      on OnFinishInput: SetBit("Interface.inputFinished")
      Appearance <- "Interface.animate"
      ObjectEnable <- "Interface.animate"
      ProcessValue <- "Interface.value"
*)

(* ===== HMI "HMI_RT_1" =====
system functions are stored by id; their names below are inferred from use

ScreenModuleEditorView "IO Field: Timer" 137x50
   IOField "Allotted Time Entry Field" at 0,0 size 137x50; FormatPattern ???????
      on OnFinishInput: SetBit("Interface.inputFinished")
      Appearance <- "Interface.animate"
      ObjectEnable <- "Interface.animate"
      ProcessValue <- "Interface.value"
*)

(* ===== HMI "HMI_RT_1" =====

ScreenModuleEditorView "LED Row" 440x28
   TextField "tfLine" at 0,0 size 110x28; Text 'Text'
      Visibility <- "interface.tfLine.visibility"
      Appearance <- "interface.tfLine.animator"
   TextField "tfTime" at 349,0 size 91x28; Text 'Text'
      Visibility <- "interface.tfTime.visibility"
      Appearance <- "interface.tfTime.animator"
   TextField "tfDropZone" at 105,0 size 42x28; Text 'Text'
      Visibility <- "interface.tfDropZone.visibility"
      Appearance <- "interface.tfDropZone.animator"
   TextField "tfSLPartNumber" at 146,0 size 209x28; Text 'Text'
      Visibility <- "interface.tfPartNumber.count"
      Appearance <- "interface.tfPartNumber.animator"
   TextField "tfDLPartNumber" at 146,0 size 209x28; Text 'Text'
      Visibility <- "interface.tfPartNumber.count"
      Appearance <- "interface.tfPartNumber.animator"
*)

(* ===== HMI "HMI_RT_1" =====
system functions are stored by id; their names below are inferred from use

ScreenModuleEditorView "Line Label" 267x40
   IOField "Line" at 86,0 size 181x40; FormatPattern ?????????
      on OnFinishInput: SetBit("interface.inputFinished")
      Appearance <- "interface.animate.ioField"
      ObjectEnable <- "interface.animate.ioField"
      Visibility <- "interface.animate.ioField"
      ProcessValue <- "interface.value"
   TextField "Line Label" at 0,0 size 267x40; Text 'Line:'
      Visibility <- "interface.animate.bg"
      Appearance <- "interface.animate.bg"
*)

(* ===== HMI "HMI_RT_1" =====
system functions are stored by id; their names below are inferred from use

ScreenModuleEditorView "PB: Graphic/Text List" 65x45
   Button "Previous Station Group" at 0,0 size 65x45; TextOff 'Text'
      on Press: function_b14e0dd5("Interface.actuate", 0)
      Visibility <- "Interface.animate"
      ObjectEnable <- "Interface.animate"
      Appearance <- "Interface.animate"
*)

(* ===== HMI "HMI_RT_1" =====
system functions are stored by id; their names below are inferred from use

ScreenModuleEditorView "PB: KP8 Button Select (Text Label)" 68x66
   Button "Station Select" at 0,0 size 68x66; TextOff 'Text'
      on Press: function_b14e0dd5("Interface.actuate", 0)
      Appearance <- "Interface.animate"
*)

(* ===== HMI "HMI_RT_1" =====

ScreenModuleEditorView "PB: KP8 Reset Button (Text Label" 68x66
   Button "Station Select" at 0,0 size 68x66; TextOff 'RESET SELECTED'
      Appearance <- "Interface.animate"
*)

(* ===== HMI "HMI_RT_1" =====

ScreenModuleEditorView "PB: KP8 Stop Runtime (Text Label)" 68x66
   Button "Station Select" at 0,0 size 68x66; TextOff 'STOP RUNTIME'
      Appearance <- "Interface.animate"
*)

(* ===== HMI "HMI_RT_1" =====
system functions are stored by id; their names below are inferred from use

ScreenModuleEditorView "PB: Station Select (Text Label)" 205x65
   Button "Station Select" at 0,0 size 205x65; TextOff 'Text'
      on Press: function_b14e0dd5("Interface.actuate", 0)
      Appearance <- "Interface.animate"
*)

(* ===== HMI "HMI_RT_1" =====
system functions are stored by id; their names below are inferred from use

ScreenModuleEditorView "PB: Text Label" 274x45
   Button "Select All Stations" at 0,0 size 274x45; TextOff 'Text'
      on Press: function_b14e0dd5("Interface.actuate", 0)
      Appearance <- "Interface.animate"
*)

(* ===== HMI "HMI_RT_1" =====
system functions are stored by id; their names below are inferred from use

ScreenModuleEditorView "Station Assignment: Button Details" 513x74
   TextField "Button Label" at 0,0 size 75x74; Text 'Text'
      Visibility <- "Interface.label.animate"
      Appearance <- "Interface.label.animate"
   TextField "Critical Time" at 70,37 size 122x37; Text 'Text'
      Visibility <- "Interface.critical.animate"
      Appearance <- "Interface.critical.animate"
   TextField "Alloted Time" at 70,0 size 122x38; Text 'Text'
      Visibility <- "Interface.alloted.animate"
      Appearance <- "Interface.alloted.animate"
   TextField "Part Number" at 185,0 size 328x74; Text 'Text'
      Visibility <- "Interface.partNumber.animate"
      Appearance <- "Interface.partNumber.animate"
   Button "Select PB" at 0,0 size 513x74; TextOff 'Text'
      on Press: function_b14e0dd5("Interface.select.actuate", 0)
      Visibility <- "Interface.select.animate"
      ObjectEnable <- "Interface.select.animate"
*)

(* ===== HMI "HMI_RT_1" =====
system functions are stored by id; their names below are inferred from use

ScreenModuleEditorView "Table Row" 1312x52
   TextField "tfLine" at 5,1 size 216x48; Text 'Text'
      Visibility <- "interface.tfLine.visibility"
      Appearance <- "interface.tfLine.animator"
   TextField "tfTime" at 1085,1 size 222x48; Text 'Text'
      Visibility <- "interface.tfTime.visibility"
      Appearance <- "interface.tfTime.animator"
   TextField "tfDropZone" at 211,1 size 236x48; Text 'Text'
      Visibility <- "interface.tfDropZone.visibility"
      Appearance <- "interface.tfDropZone.animator"
   TextField "tfSLPartNumber" at 445,1 size 650x48; Text 'Text'
      Visibility <- "interface.tfPartNumber.count"
      Appearance <- "interface.tfPartNumber.animator"
   Button "pbSelect" at 0,0 size 1312x52; TextOff 'Text'
      on Release: ResetBit("interface.pbSelection.request")
      on Press: SetBit("interface.pbSelection.request")
      Visibility <- "interface.pbSelection.visibility"
   Rectangle "rtBackground" at 0,0 size 1312x52
      Visibility <- "interface.rtBackground.visibility"
   TextField "tfDLPartNumber" at 445,1 size 650x48; Text 'Text'
      Visibility <- "interface.tfPartNumber.count"
      Appearance <- "interface.tfPartNumber.animator"
*)

(* ===== HMI "HMI_RT_1" =====
system functions are stored by id; their names below are inferred from use

ScreenModuleEditorView "PB: Text Label" 274x45
   Button "Select All Stations" at 0,0 size 274x45; TextOff 'Text'
      on Press: function_b14e0dd5("Interface.actuate", 0)
      Appearance <- "Interface.animate"
      ObjectEnable <- "Interface.animate"
*)

(* ===== HMI "HMI_RT_1" =====
system functions are stored by id; their names below are inferred from use

ScreenModuleEditorView "PB: KP8 Button Select (Text Label)" 68x66
   Button "Station Select" at 0,0 size 68x66; TextOff 'Text'
      on Press: function_b14e0dd5("Interface.actuate", 0)
      Appearance <- "Interface.animate"
      ObjectEnable <- "Interface.animate"
*)

(* ===== HMI "HMI_RT_1" =====
system functions are stored by id; their names below are inferred from use

ScreenModuleEditorView "PB: KP8 Reset Button (Text Label" 68x66
   Button "Station Select" at 0,0 size 68x66; TextOff 'RESET SELECTED'
      Appearance <- "Interface.animate"
      on Press: function_b14e0dd5("Interface.actuate", 0)
*)